FUNCTION_BLOCK AUDI2_TO_AUDI (* Composite FB for convert bidirectional AUDI2 to unidirectional AUDI *)
  (* Standard: 61499-2; Function: AUDI2_BIDIR forwards its incoming (EO1) side out as a plain unidirectional signal via AUDI_OUT. AUDI_IN publishes its value onto the outgoing (EI1) side of AUDI2_BIDIR.; Description: Copyright (c) 2026 HR Agrartechnik GmbH This program and the accompanying materials are made available under the terms of the Eclipse Public License 2.0 which is available at https://www.eclipse.org/legal/epl-2.0/ SPDX-License-Identifier: EPL-2.0 *)
  (* Version 1.0, 2026-09-12, Franz Höpfinger, HR Agrartechnik GmbH, Initial Version - Konvertierungsfamilie vervollstaendigt (analog zu AR2/AB2/AE2). *)
  PACKAGE adapter::conversion::bidirectional;
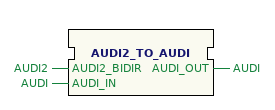
  SOCKETS
    AUDI2_BIDIR : adapter::types::bidirectional::AUDI2; (* Adapter Input: bidirectional tap, incoming side forwarded to AUDI_OUT, outgoing side driven by AUDI_IN *)
    AUDI_IN : adapter::types::unidirectional::AUDI; (* Adapter Input: unidirectional source *)
  END_SOCKETS
  PLUGS
    AUDI_OUT : adapter::types::unidirectional::AUDI; (* Adapter Output: mirrors AUDI2_BIDIR's incoming (indication) side *)
  END_PLUGS
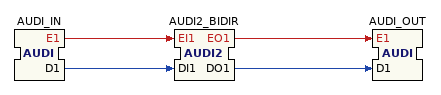
  EVENT_CONNECTIONS
    AUDI2_BIDIR.EO1 TO AUDI_OUT.E1;
    AUDI_IN.E1 TO AUDI2_BIDIR.EI1;
  END_CONNECTIONS
  DATA_CONNECTIONS
    AUDI2_BIDIR.DO1 TO AUDI_OUT.D1;
    AUDI_IN.D1 TO AUDI2_BIDIR.DI1;
  END_CONNECTIONS
END_FUNCTION_BLOCK
